{attribute 'qualified_only'}
VAR_GLOBAL
	{attribute 'OPC.UA.DA' := '1'}
	StationParameter: STRING;
	{attribute 'OPC.UA.DA' := '1'}
	StationValue: STRING;
	inPos1: INT;
	inPos2: INT;
	pistLock: INT;
END_VAR

(* stored: Version 1.1.0.1, ProductVersion 3.1.4024.5
   GVL OPCVAR: Id {fd6c5c14-43a4-46a0-952e-b1336be2922b} *)
